TYPE DUT_VALVE :
STRUCT
	Cs: DUT_CS;
	Hmi: DUT_HMI;
	Sts: DUT_STS;
	Alm: DUT_ALM;
END_STRUCT
END_TYPE

(* stored: Version 1.1.0.1, ProductVersion 3.1.4024.12
   DUT DUT_VALVE: Id {7768549f-516b-48d9-ba55-440da92000e0} *)
